// Mitsubishi GX Works2 project: 미니프로젝트6   PLC: Q03UDV

PROGRAM MAIN
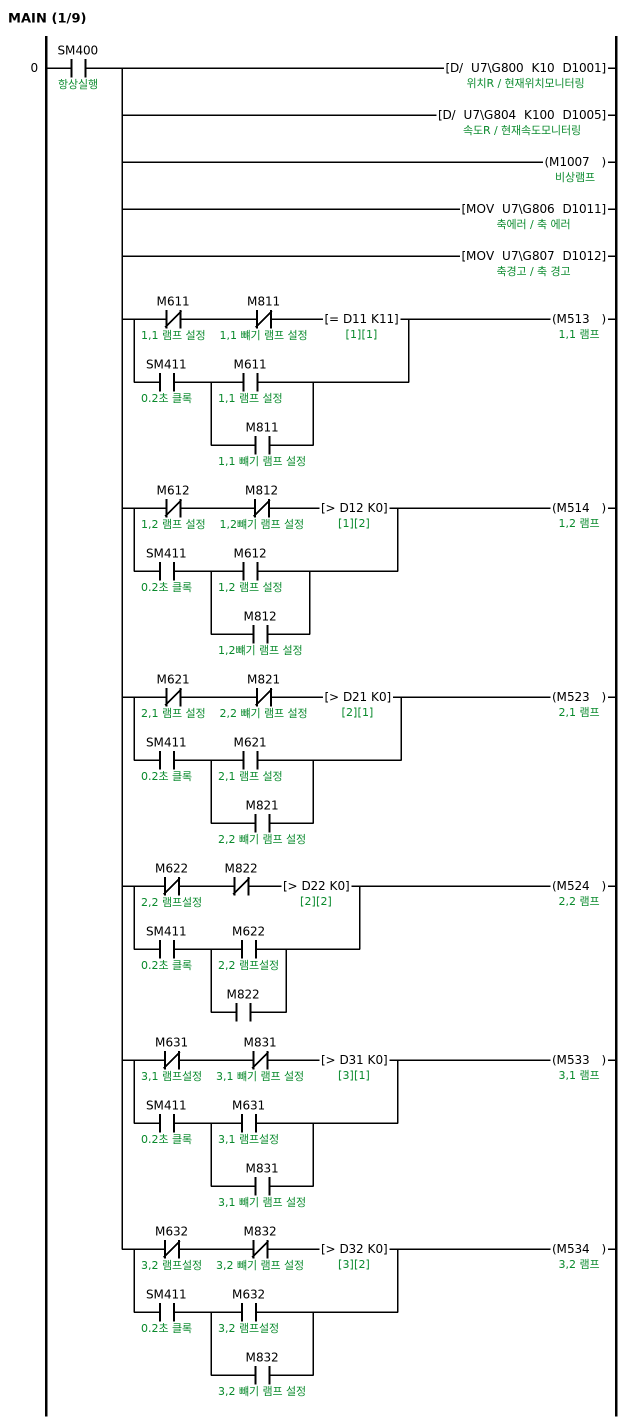
0     LD      SM400  ; 항상실행
      D/      U7\G800 K10 D1001  ; 위치R / 현재위치모니터링
      D/      U7\G804 K100 D1005  ; 속도R / 현재속도모니터링
      OUT     M1007  ; 비상램프
      MOV     U7\G806 D1011  ; 축에러 / 축 에러
      MOV     U7\G807 D1012  ; 축경고 / 축 경고
      MPS
      LDI     M611  ; 1,1 램프 설정
      ANI     M811  ; 1,1 뺴기 램프 설정
      AND=    D11 K11  ; [1][1]
      LD      SM411  ; 0.2초 클록
      LD      M611  ; 1,1 램프 설정
      OR      M811  ; 1,1 뺴기 램프 설정
      ANB
      ORB
      ANB
      OUT     M513  ; 1,1 램프
      MRD
      LDI     M612  ; 1,2 램프 설정
      ANI     M812  ; 1,2뺴기 램프 설정
      AND>    D12 K0  ; [1][2]
      LD      SM411  ; 0.2초 클록
      LD      M612  ; 1,2 램프 설정
      OR      M812  ; 1,2뺴기 램프 설정
      ANB
      ORB
      ANB
      OUT     M514  ; 1,2 램프
      MRD
      LDI     M621  ; 2,1 램프 설정
      ANI     M821  ; 2,2 뺴기 램프 설정
      AND>    D21 K0  ; [2][1]
      LD      SM411  ; 0.2초 클록
      LD      M621  ; 2,1 램프 설정
      OR      M821  ; 2,2 뺴기 램프 설정
      ANB
      ORB
      ANB
      OUT     M523  ; 2,1 램프
      MRD
      LDI     M622  ; 2,2 램프설정
      ANI     M822
      AND>    D22 K0  ; [2][2]
      LD      SM411  ; 0.2초 클록
      LD      M622  ; 2,2 램프설정
      OR      M822
      ANB
      ORB
      ANB
      OUT     M524  ; 2,2 램프
      MRD
      LDI     M631  ; 3,1 램프설정
      ANI     M831  ; 3,1 뺴기 램프 설정
      AND>    D31 K0  ; [3][1]
      LD      SM411  ; 0.2초 클록
      LD      M631  ; 3,1 램프설정
      OR      M831  ; 3,1 뺴기 램프 설정
      ANB
      ORB
      ANB
      OUT     M533  ; 3,1 램프
      MPP
      LDI     M632  ; 3,2 램프설정
      ANI     M832  ; 3,2 뺴기 램프 설정
      AND>    D32 K0  ; [3][2]
      LD      SM411  ; 0.2초 클록
      LD      M632  ; 3,2 램프설정
      OR      M832  ; 3,2 뺴기 램프 설정
      ANB
      ORB
      ANB
      OUT     M534  ; 3,2 램프
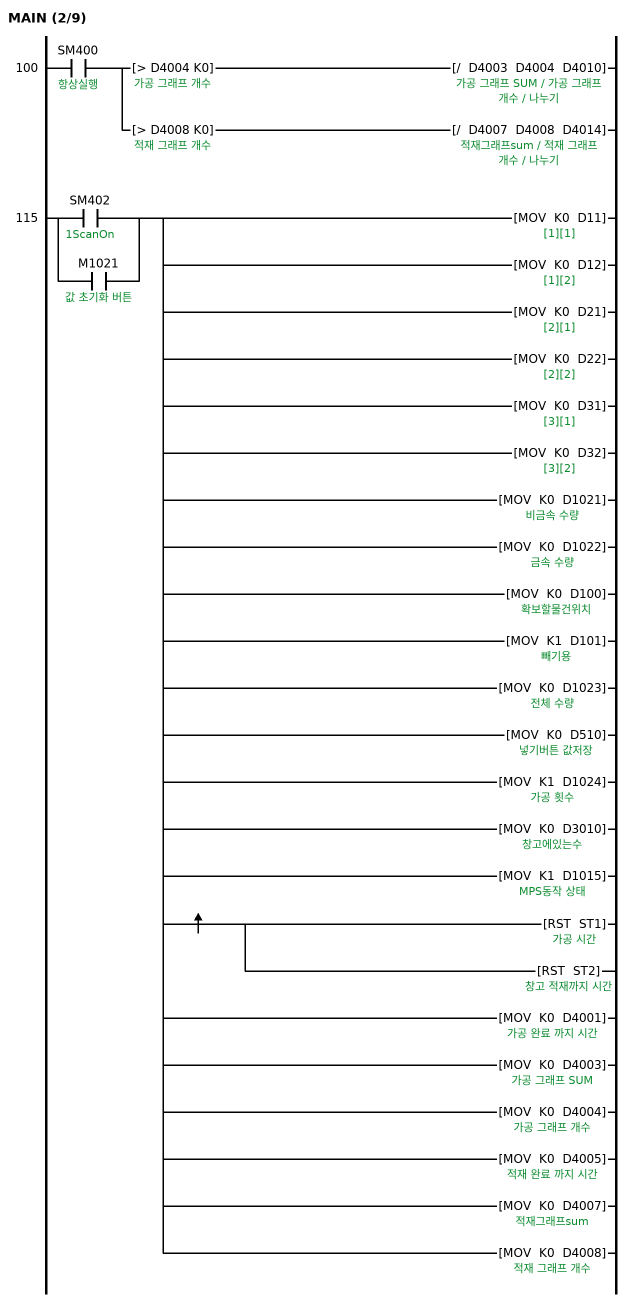
100   LD      SM400  ; 항상실행
      MPS
      AND>    D4004 K0  ; 가공 그래프 개수
      /       D4003 D4004 D4010  ; 가공 그래프 SUM / 나누기
      MPP
      AND>    D4008 K0  ; 적재 그래프 개수
      /       D4007 D4008 D4014  ; 적재그래프sum / 나누기
115   LD      SM402  ; 1ScanOn
      OR      M1021  ; 값 초기화 버튼
      MOV     K0 D11
      MOV     K0 D12
      MOV     K0 D21
      MOV     K0 D22
      MOV     K0 D31
      MOV     K0 D32
      MOV     K0 D1021  ; 비금속 수량
      MOV     K0 D1022  ; 금속 수량
      MOV     K0 D100  ; 확보할물건위치
      MOV     K1 D101  ; 빼기용
      MOV     K0 D1023  ; 전체 수량
      MOV     K0 D510  ; 넣기버튼 값저장
      MOV     K1 D1024  ; 가공 횟수
      MOV     K0 D3010  ; 창고에있는수
      MOV     K1 D1015  ; MPS동작 상태
      MPS
      MEP
      RST     ST1  ; 가공 시간
      RST     ST2  ; 창고 적재까지 시간
      MPP
      MOV     K0 D4001  ; 가공 완료 까지 시간
      MOV     K0 D4003
      MOV     K0 D4004
      MOV     K0 D4005  ; 적재 완료 까지 시간
      MOV     K0 D4007
      MOV     K0 D4008
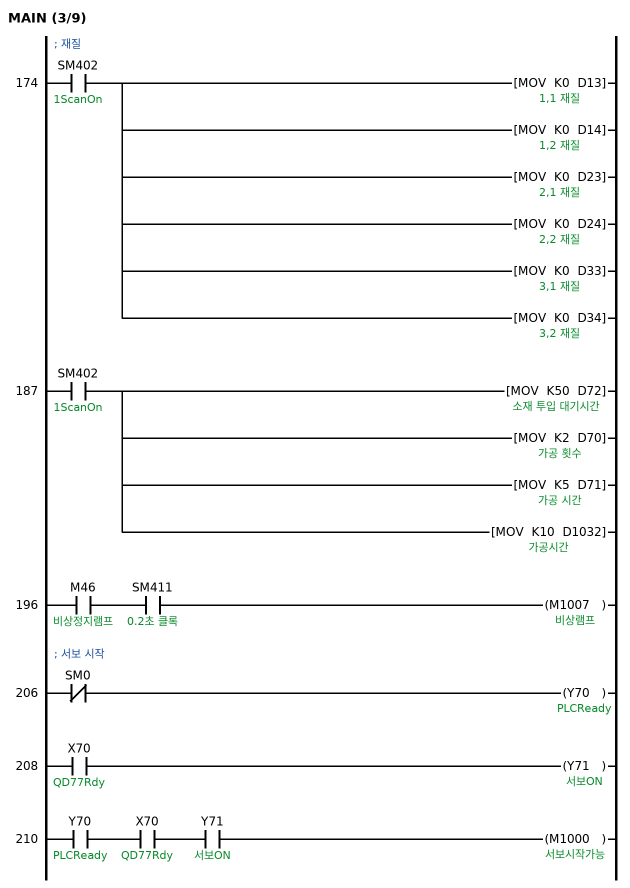
; 재질
174   LD      SM402  ; 1ScanOn
      MOV     K0 D13  ; 1,1 재질
      MOV     K0 D14  ; 1,2 재질
      MOV     K0 D23  ; 2,1 재질
      MOV     K0 D24  ; 2,2 재질
      MOV     K0 D33  ; 3,1 재질
      MOV     K0 D34  ; 3,2 재질
187   LD      SM402  ; 1ScanOn
      MOV     K50 D72  ; 소재 투입 대기시간
      MOV     K2 D70  ; 가공 횟수
      MOV     K5 D71  ; 가공 시간
      MOV     K10 D1032  ; 가공시간
196   LD      M46  ; 비상정지램프
      AND     SM411  ; 0.2초 클록
      OUT     M1007  ; 비상램프
; 서보 시작
206   LDI     SM0
      OUT     Y70  ; PLCReady
208   LD      X70  ; QD77Rdy
      OUT     Y71  ; 서보ON
210   LD      Y70  ; PLCReady
      AND     X70  ; QD77Rdy
      AND     Y71  ; 서보ON
      OUT     M1000  ; 서보시작가능
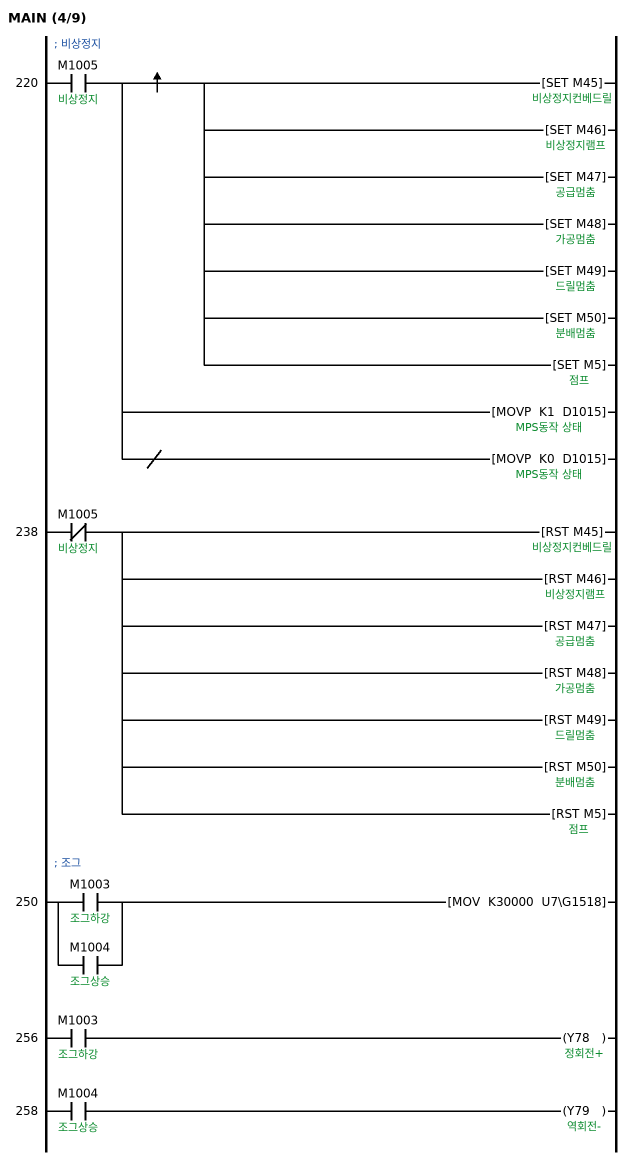
; 비상정지
220   LD      M1005  ; 비상정지
      MPS
      MEP
      SET     M45  ; 비상정지컨베드릴
      SET     M46  ; 비상정지램프
      SET     M47  ; 공급멈춤
      SET     M48  ; 가공멈춤
      SET     M49  ; 드릴멈춤
      SET     M50  ; 분배멈춤
      SET     M5  ; 점프
      MPP
      MOVP    K1 D1015
      INV
      MOVP    K0 D1015
238   LDI     M1005  ; 비상정지
      RST     M45  ; 비상정지컨베드릴
      RST     M46  ; 비상정지램프
      RST     M47  ; 공급멈춤
      RST     M48  ; 가공멈춤
      RST     M49  ; 드릴멈춤
      RST     M50  ; 분배멈춤
      RST     M5  ; 점프
; 조그
250   LD      M1003  ; 조그하강
      OR      M1004  ; 조그상승
      MOV     K30000 U7\G1518
256   LD      M1003  ; 조그하강
      OUT     Y78  ; 정회전+
258   LD      M1004  ; 조그상승
      OUT     Y79  ; 역회전-
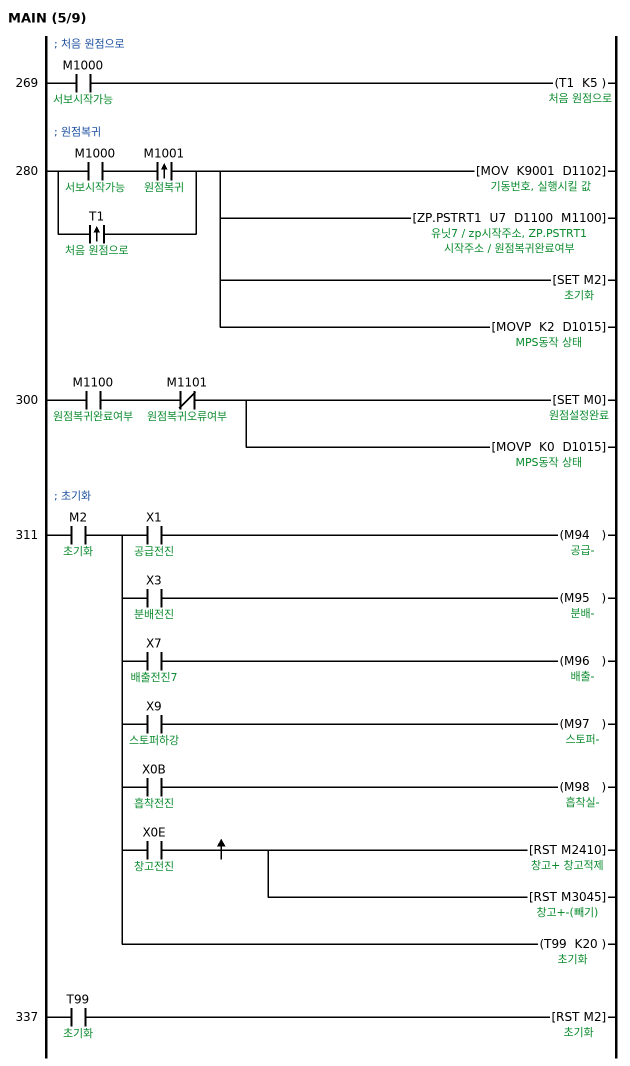
; 처음 원점으로
269   LD      M1000  ; 서보시작가능
      OUT     T1 K5  ; 처음 원점으로
; 원점복귀
280   LD      M1000  ; 서보시작가능
      ANDP    M1001  ; 원점복귀
      ORP     T1  ; 처음 원점으로
      MOV     K9001 D1102  ; 기동번호, 실행시킬 값
      ZP.PSTRT1 U7 D1100 M1100  ; 유닛7 / zp시작주소, ZP.PSTRT1 시작주소 / 원점복귀완료여부
      SET     M2  ; 초기화
      MOVP    K2 D1015
300   LD      M1100  ; 원점복귀완료여부
      ANI     M1101  ; 원점복귀오류여부
      SET     M0  ; 원점설정완료
      MOVP    K0 D1015
; 초기화
311   LD      M2  ; 초기화
      MPS
      AND     X1  ; 공급전진
      OUT     M94  ; 공급-
      MRD
      AND     X3  ; 분배전진
      OUT     M95  ; 분배-
      MRD
      AND     X7  ; 배출전진7
      OUT     M96  ; 배출-
      MRD
      AND     X9  ; 스토퍼하강
      OUT     M97  ; 스토퍼-
      MRD
      AND     X0B  ; 흡착전진
      OUT     M98  ; 흡착실-
      MRD
      AND     X0E  ; 창고전진
      MEP
      RST     M2410  ; 창고+ 창고적제
      RST     M3045  ; 창고+-(빼기)
      MPP
      OUT     T99 K20  ; 초기화
337   LD      T99  ; 초기화
      RST     M2  ; 초기화
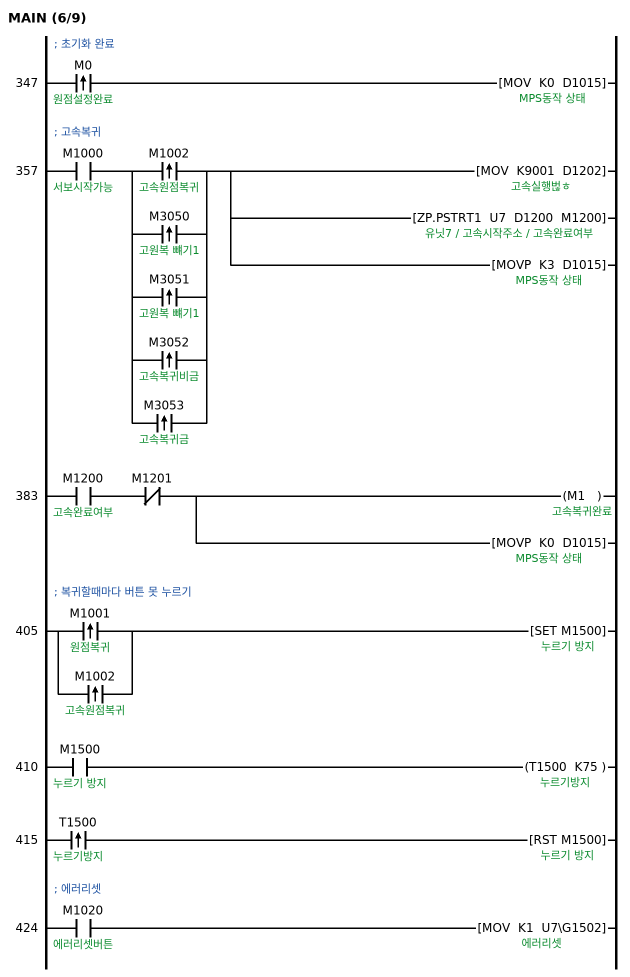
; 초기화 완료
347   LDP     M0  ; 원점설정완료
      MOV     K0 D1015
; 고속복귀
357   LD      M1000  ; 서보시작가능
      LDP     M1002  ; 고속원점복귀
      ORP     M3050  ; 고원복 뺴기1
      ORP     M3051  ; 고원복 뺴기1
      ORP     M3052  ; 고속복귀비금
      ORP     M3053  ; 고속복귀금
      ANB
      MOV     K9001 D1202  ; 고속실행벊ㅎ
      ZP.PSTRT1 U7 D1200 M1200  ; 고속시작주소 / 고속완료여부
      MOVP    K3 D1015
383   LD      M1200  ; 고속완료여부
      ANI     M1201
      OUT     M1  ; 고속복귀완료
      MOVP    K0 D1015
; 복귀할때마다 버튼 못 누르기
405   LDP     M1001  ; 원점복귀
      ORP     M1002  ; 고속원점복귀
      SET     M1500  ; 누르기 방지
410   LD      M1500  ; 누르기 방지
      OUT     T1500 K75  ; 누르기방지
415   LDP     T1500  ; 누르기방지
      RST     M1500  ; 누르기 방지
; 에러리셋
424   LD      M1020  ; 에러리셋버튼
      MOV     K1 U7\G1502  ; 에러리셋
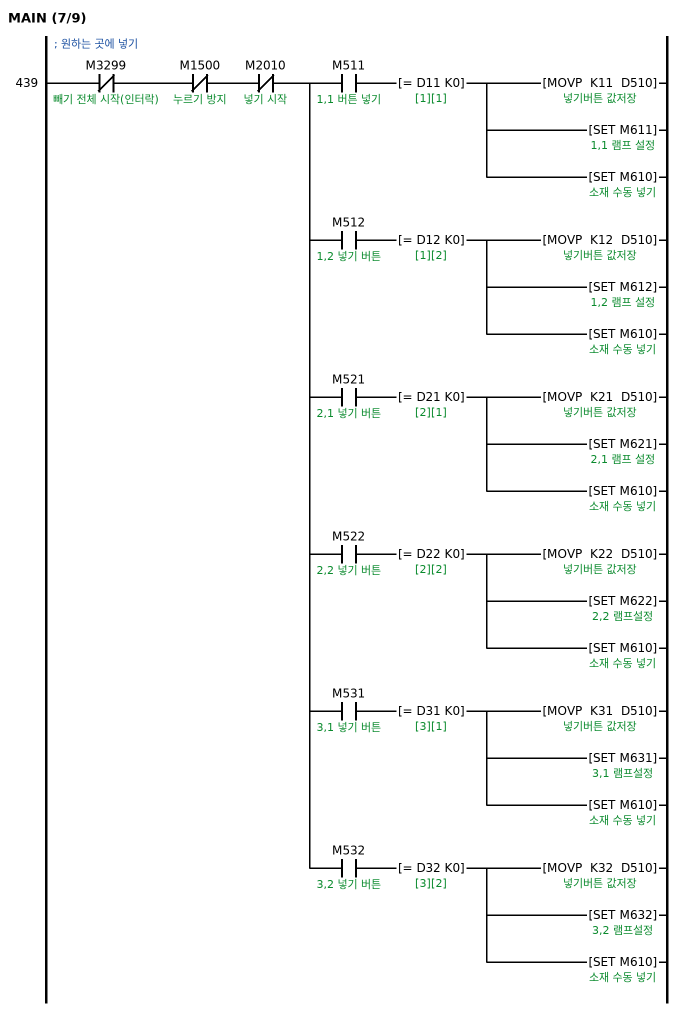
; 원하는 곳에 넣기
439   LDI     M3299  ; 빼기 전체 시작(인터락)
      ANI     M1500  ; 누르기 방지
      ANI     M2010  ; 넣기 시작
      MPS
      AND     M511  ; 1,1 버튼 넣기
      AND=    D11 K0  ; [1][1]
      MOVP    K11 D510
      SET     M611  ; 1,1 램프 설정
      SET     M610  ; 소재 수동 넣기
      MRD
      AND     M512  ; 1,2 넣기 버튼
      AND=    D12 K0  ; [1][2]
      MOVP    K12 D510
      SET     M612  ; 1,2 램프 설정
      SET     M610  ; 소재 수동 넣기
      MRD
      AND     M521  ; 2,1 넣기 버튼
      AND=    D21 K0  ; [2][1]
      MOVP    K21 D510
      SET     M621  ; 2,1 램프 설정
      SET     M610  ; 소재 수동 넣기
      MRD
      AND     M522  ; 2,2 넣기 버튼
      AND=    D22 K0  ; [2][2]
      MOVP    K22 D510
      SET     M622  ; 2,2 램프설정
      SET     M610  ; 소재 수동 넣기
      MRD
      AND     M531  ; 3,1 넣기 버튼
      AND=    D31 K0  ; [3][1]
      MOVP    K31 D510
      SET     M631  ; 3,1 램프설정
      SET     M610  ; 소재 수동 넣기
      MPP
      AND     M532  ; 3,2 넣기 버튼
      AND=    D32 K0  ; [3][2]
      MOVP    K32 D510
      SET     M632  ; 3,2 램프설정
      SET     M610  ; 소재 수동 넣기
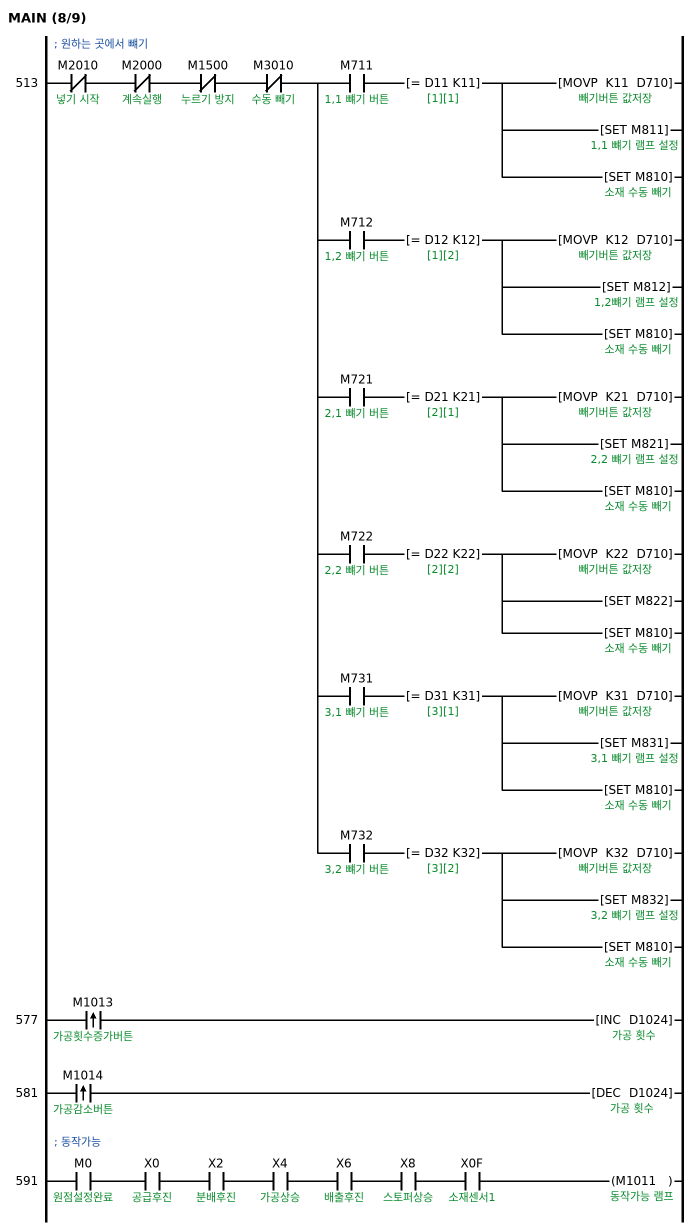
; 원하는 곳에서 뺴기
513   LDI     M2010  ; 넣기 시작
      ANI     M2000  ; 계속실행
      ANI     M1500  ; 누르기 방지
      ANI     M3010  ; 수동 빼기
      MPS
      AND     M711  ; 1,1 뺴기 버튼
      AND=    D11 K11  ; [1][1]
      MOVP    K11 D710  ; 빼기버튼 값저장
      SET     M811  ; 1,1 뺴기 램프 설정
      SET     M810  ; 소재 수동 빼기
      MRD
      AND     M712  ; 1,2 뺴기 버튼
      AND=    D12 K12  ; [1][2]
      MOVP    K12 D710
      SET     M812  ; 1,2뺴기 램프 설정
      SET     M810  ; 소재 수동 빼기
      MRD
      AND     M721  ; 2,1 뺴기 버튼
      AND=    D21 K21  ; [2][1]
      MOVP    K21 D710
      SET     M821  ; 2,2 뺴기 램프 설정
      SET     M810  ; 소재 수동 빼기
      MRD
      AND     M722  ; 2,2 뺴기 버튼
      AND=    D22 K22  ; [2][2]
      MOVP    K22 D710
      SET     M822
      SET     M810  ; 소재 수동 빼기
      MRD
      AND     M731  ; 3,1 뺴기 버튼
      AND=    D31 K31  ; [3][1]
      MOVP    K31 D710
      SET     M831  ; 3,1 뺴기 램프 설정
      SET     M810  ; 소재 수동 빼기
      MPP
      AND     M732  ; 3,2 뺴기 버튼
      AND=    D32 K32  ; [3][2]
      MOVP    K32 D710
      SET     M832  ; 3,2 뺴기 램프 설정
      SET     M810  ; 소재 수동 빼기
577   LDP     M1013  ; 가공횟수증가버튼
      INC     D1024
581   LDP     M1014  ; 가공감소버튼
      DEC     D1024
; 동작가능
591   LD      M0  ; 원점설정완료
      AND     X0  ; 공급후진
      AND     X2  ; 분배후진
      AND     X4  ; 가공상승
      AND     X6  ; 배출후진
      AND     X8  ; 스토퍼상승
      AND     X0F  ; 소재센서1
      OUT     M1011  ; 동작가능 램프
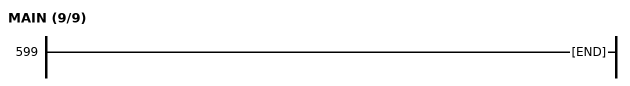
599   END
END_PROGRAM

PROGRAM OUTPUT
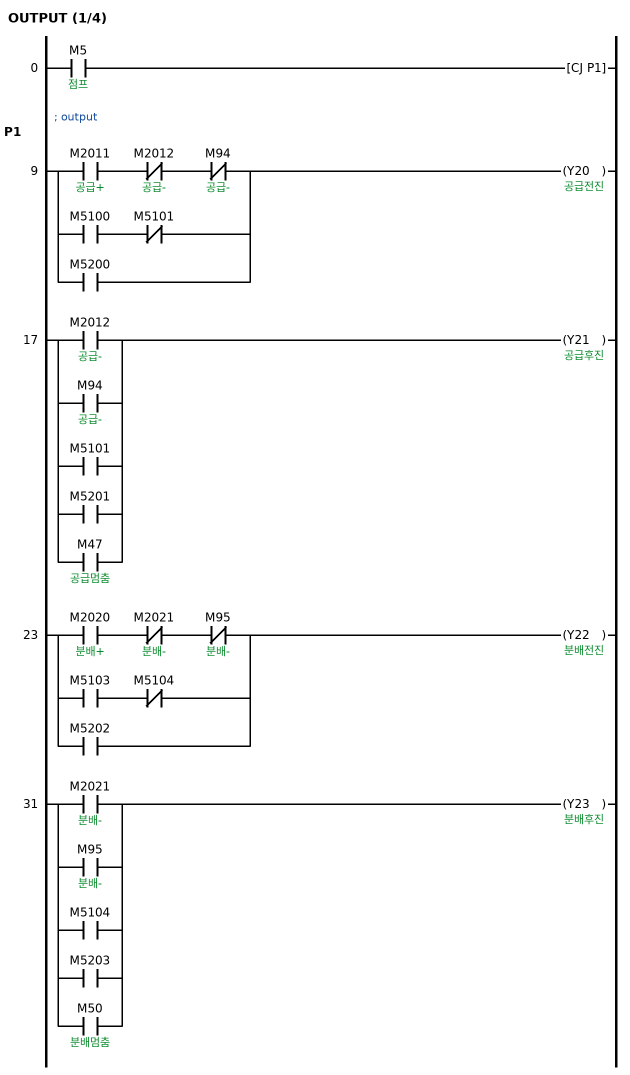
0     LD      M5  ; 점프
      CJ      P1
; output
      P1
9     LD      M2011  ; 공급+
      ANI     M2012  ; 공급-
      ANI     M94  ; 공급-
      LD      M5100
      ANI     M5101
      ORB
      OR      M5200
      OUT     Y20  ; 공급전진
17    LD      M2012  ; 공급-
      OR      M94  ; 공급-
      OR      M5101
      OR      M5201
      OR      M47  ; 공급멈춤
      OUT     Y21  ; 공급후진
23    LD      M2020  ; 분배+
      ANI     M2021  ; 분배-
      ANI     M95  ; 분배-
      LD      M5103
      ANI     M5104
      ORB
      OR      M5202
      OUT     Y22  ; 분배전진
31    LD      M2021  ; 분배-
      OR      M95  ; 분배-
      OR      M5104
      OR      M5203
      OR      M50  ; 분배멈춤
      OUT     Y23  ; 분배후진
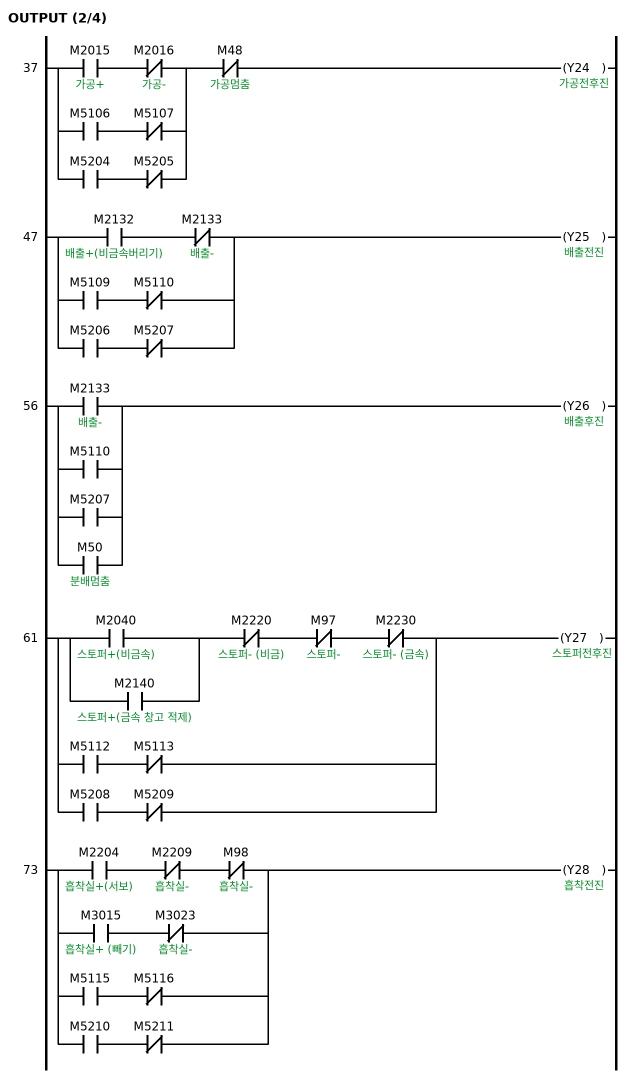
37    LD      M2015  ; 가공+
      ANI     M2016  ; 가공-
      LD      M5106
      ANI     M5107
      ORB
      LD      M5204
      ANI     M5205
      ORB
      ANI     M48  ; 가공멈춤
      OUT     Y24  ; 가공전후진
47    LD      M2132  ; 배출+(비금속버리기)
      ANI     M2133  ; 배출-
      LD      M5109
      ANI     M5110
      ORB
      LD      M5206
      ANI     M5207
      ORB
      OUT     Y25  ; 배출전진
56    LD      M2133  ; 배출-
      OR      M5110
      OR      M5207
      OR      M50  ; 분배멈춤
      OUT     Y26  ; 배출후진
61    LD      M2040  ; 스토퍼+(비금속)
      OR      M2140  ; 스토퍼+(금속 창고 적제)
      ANI     M2220  ; 스토퍼- (비금)
      ANI     M97  ; 스토퍼-
      ANI     M2230  ; 스토퍼- (금속)
      LD      M5112
      ANI     M5113
      ORB
      LD      M5208
      ANI     M5209
      ORB
      OUT     Y27  ; 스토퍼전후진
73    LD      M2204  ; 흡착실+(서보)
      ANI     M2209  ; 흡착실-
      ANI     M98  ; 흡착실-
      LD      M3015  ; 흡착실+ (빼기)
      ANI     M3023  ; 흡착실-
      ORB
      LD      M5115
      ANI     M5116
      ORB
      LD      M5210
      ANI     M5211
      ORB
      OUT     Y28  ; 흡착전진
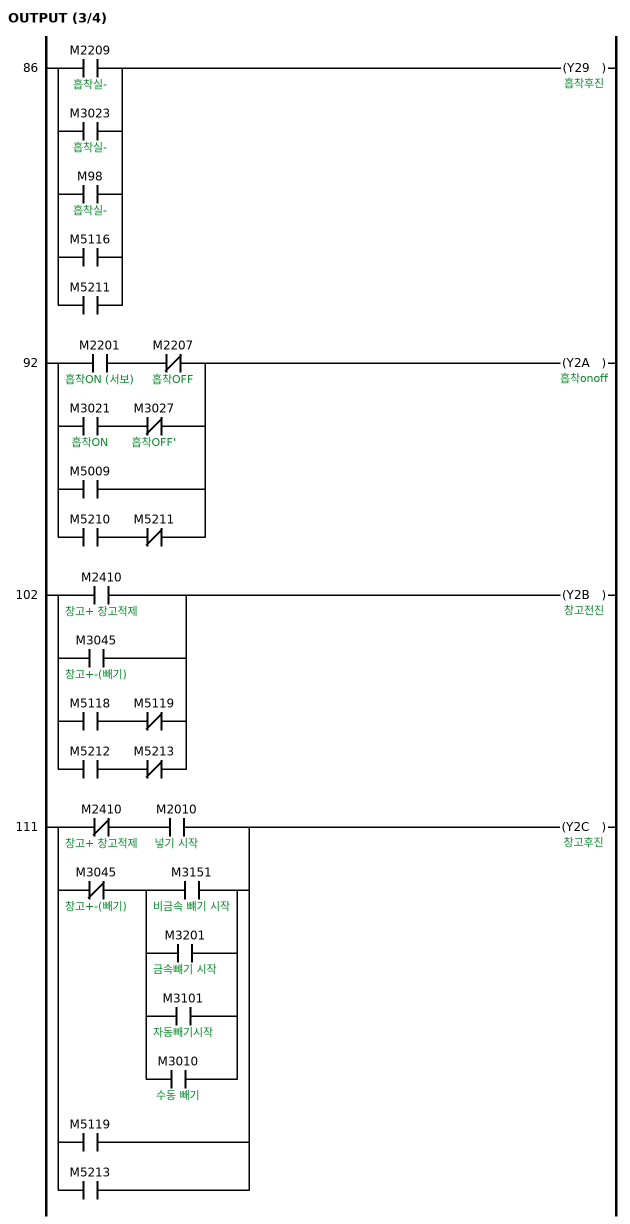
86    LD      M2209  ; 흡착실-
      OR      M3023  ; 흡착실-
      OR      M98  ; 흡착실-
      OR      M5116
      OR      M5211
      OUT     Y29  ; 흡착후진
92    LD      M2201  ; 흡착ON (서보)
      ANI     M2207  ; 흡착OFF
      LD      M3021  ; 흡착ON
      ANI     M3027  ; 흡착OFF'
      ORB
      OR      M5009
      LD      M5210
      ANI     M5211
      ORB
      OUT     Y2A  ; 흡착onoff
102   LD      M2410  ; 창고+ 창고적제
      OR      M3045  ; 창고+-(빼기)
      LD      M5118
      ANI     M5119
      ORB
      LD      M5212
      ANI     M5213
      ORB
      OUT     Y2B  ; 창고전진
111   LDI     M2410  ; 창고+ 창고적제
      AND     M2010  ; 넣기 시작
      LDI     M3045  ; 창고+-(빼기)
      LD      M3151  ; 비금속 뺴기 시작
      OR      M3201  ; 금속뺴기 시작
      OR      M3101  ; 자동빼기시작
      OR      M3010  ; 수동 빼기
      ANB
      ORB
      OR      M5119
      OR      M5213
      OUT     Y2C  ; 창고후진
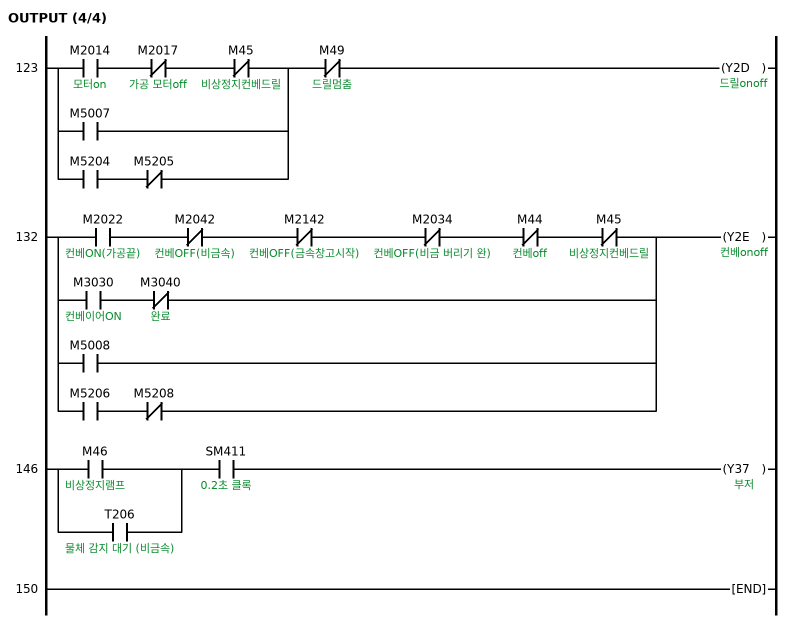
123   LD      M2014  ; 모터on
      ANI     M2017  ; 가공 모터off
      ANI     M45  ; 비상정지컨베드릴
      OR      M5007
      LD      M5204
      ANI     M5205
      ORB
      ANI     M49  ; 드릴멈춤
      OUT     Y2D  ; 드릴onoff
132   LD      M2022  ; 컨베ON(가공끝)
      ANI     M2042  ; 컨베OFF(비금속)
      ANI     M2142  ; 컨베OFF(금속창고시작)
      ANI     M2034  ; 컨베OFF(비금 버리기 완)
      ANI     M44  ; 컨베off
      ANI     M45  ; 비상정지컨베드릴
      LD      M3030  ; 컨베이어ON
      ANI     M3040  ; 완료
      ORB
      OR      M5008
      LD      M5206
      ANI     M5208
      ORB
      OUT     Y2E  ; 컨베onoff
146   LD      M46  ; 비상정지램프
      OR      T206  ; 물체 감지 대기 (비금속)
      AND     SM411  ; 0.2초 클록
      OUT     Y37  ; 부저
150   END
END_PROGRAM

PROGRAM LOADING
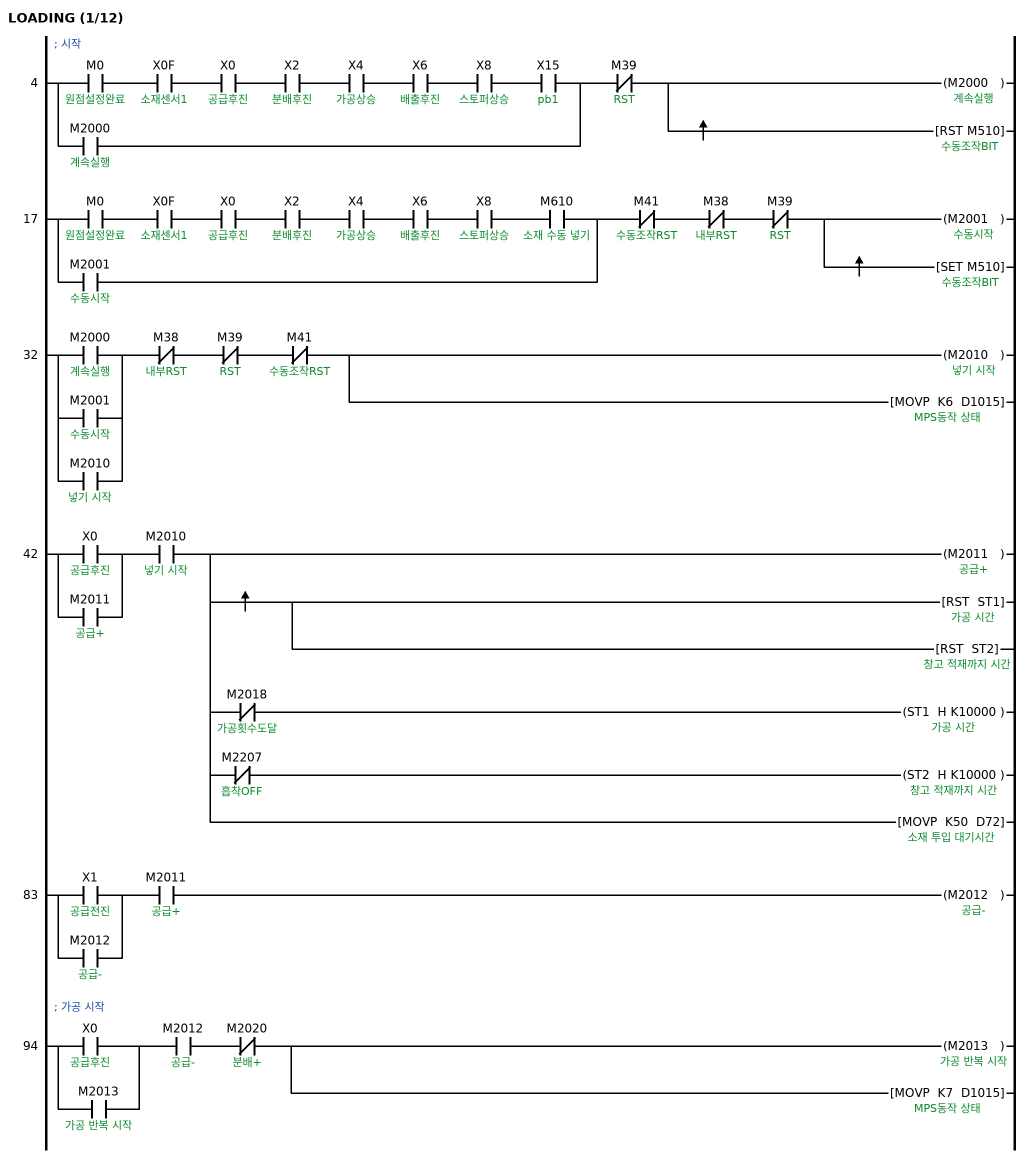
; 시작
4     LD      M0  ; 원점설정완료
      AND     X0F  ; 소재센서1
      AND     X0  ; 공급후진
      AND     X2  ; 분배후진
      AND     X4  ; 가공상승
      AND     X6  ; 배출후진
      AND     X8  ; 스토퍼상승
      AND     X15  ; pb1
      OR      M2000  ; 계속실행
      ANI     M39  ; RST
      OUT     M2000  ; 계속실행
      MEP
      RST     M510  ; 수동조작BIT
17    LD      M0  ; 원점설정완료
      AND     X0F  ; 소재센서1
      AND     X0  ; 공급후진
      AND     X2  ; 분배후진
      AND     X4  ; 가공상승
      AND     X6  ; 배출후진
      AND     X8  ; 스토퍼상승
      AND     M610  ; 소재 수동 넣기
      OR      M2001  ; 수동시작
      ANI     M41  ; 수동조작RST
      ANI     M38  ; 내부RST
      ANI     M39  ; RST
      OUT     M2001  ; 수동시작
      MEP
      SET     M510  ; 수동조작BIT
32    LD      M2000  ; 계속실행
      OR      M2001  ; 수동시작
      OR      M2010  ; 넣기 시작
      ANI     M38  ; 내부RST
      ANI     M39  ; RST
      ANI     M41  ; 수동조작RST
      OUT     M2010  ; 넣기 시작
      MOVP    K6 D1015  ; MPS동작 상태
42    LD      X0  ; 공급후진
      OR      M2011  ; 공급+
      AND     M2010  ; 넣기 시작
      OUT     M2011  ; 공급+
      MPS
      MEP
      RST     ST1  ; 가공 시간
      RST     ST2  ; 창고 적재까지 시간
      MRD
      ANI     M2018  ; 가공횟수도달
      OUTH    ST1 K10000  ; 가공 시간
      MRD
      ANI     M2207  ; 흡착OFF
      OUTH    ST2 K10000  ; 창고 적재까지 시간
      MPP
      MOVP    K50 D72  ; 소재 투입 대기시간
        [note] 5초대기시간 초기화
83    LD      X1  ; 공급전진
      OR      M2012  ; 공급-
      AND     M2011  ; 공급+
      OUT     M2012  ; 공급-
; 가공 시작
94    LD      X0  ; 공급후진
      OR      M2013  ; 가공 반복 시작
      AND     M2012  ; 공급-
      ANI     M2020  ; 분배+
      OUT     M2013  ; 가공 반복 시작
      MOVP    K7 D1015
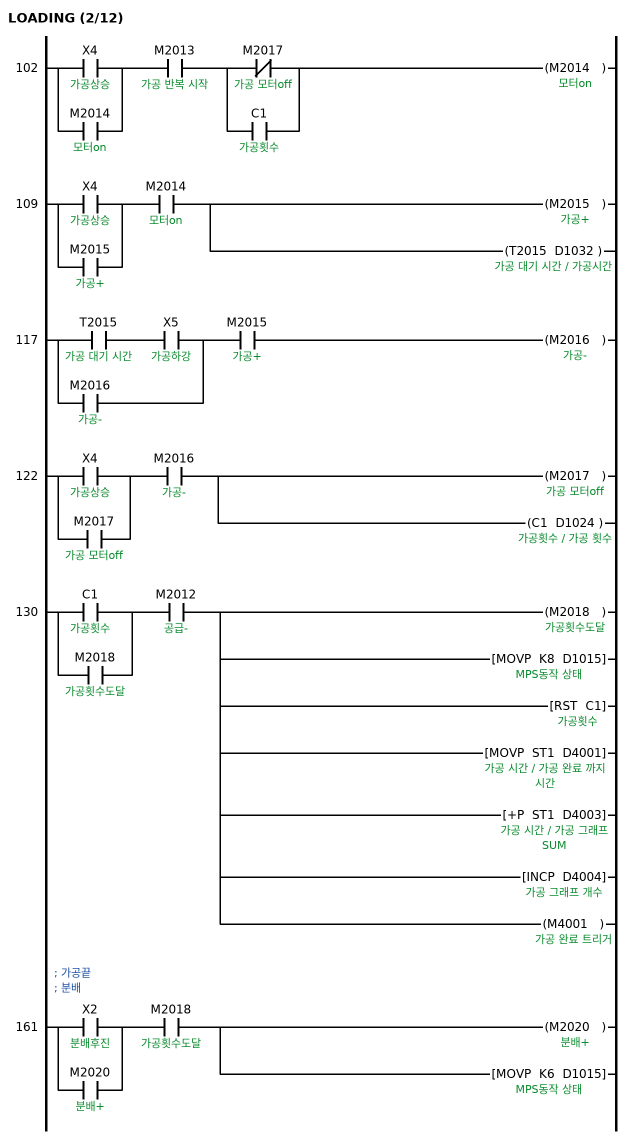
102   LD      X4  ; 가공상승
      OR      M2014  ; 모터on
      AND     M2013  ; 가공 반복 시작
      LDI     M2017  ; 가공 모터off
      OR      C1  ; 가공횟수
      ANB
      OUT     M2014  ; 모터on
109   LD      X4  ; 가공상승
      OR      M2015  ; 가공+
      AND     M2014  ; 모터on
      OUT     M2015  ; 가공+
      OUT     T2015 D1032  ; 가공 대기 시간 / 가공시간
117   LD      T2015  ; 가공 대기 시간
      AND     X5  ; 가공하강
      OR      M2016  ; 가공-
      AND     M2015  ; 가공+
      OUT     M2016  ; 가공-
122   LD      X4  ; 가공상승
      OR      M2017  ; 가공 모터off
      AND     M2016  ; 가공-
      OUT     M2017  ; 가공 모터off
      OUT     C1 D1024  ; 가공횟수 / 가공 횟수
130   LD      C1  ; 가공횟수
      OR      M2018  ; 가공횟수도달
      AND     M2012  ; 공급-
      OUT     M2018  ; 가공횟수도달
      MOVP    K8 D1015
      RST     C1  ; 가공횟수
      MOVP    ST1 D4001  ; 가공 완료 까지 시간
      +P      ST1 D4003  ; 가공 그래프 SUM
      INCP    D4004  ; 가공 그래프 개수
      OUT     M4001  ; 가공 완료 트리거
; 가공끝
; 분배
161   LD      X2  ; 분배후진
      OR      M2020  ; 분배+
      AND     M2018  ; 가공횟수도달
      OUT     M2020  ; 분배+
      MOVP    K6 D1015
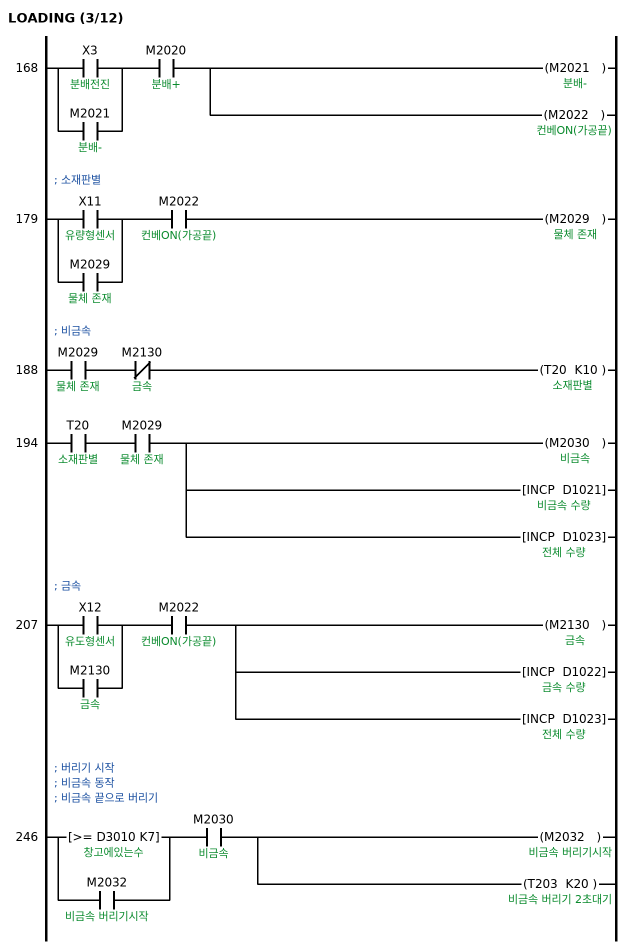
168   LD      X3  ; 분배전진
      OR      M2021  ; 분배-
      AND     M2020  ; 분배+
      OUT     M2021  ; 분배-
      OUT     M2022  ; 컨베ON(가공끝)
; 소재판별
179   LD      X11  ; 유량형센서
      OR      M2029  ; 물체 존재
      AND     M2022  ; 컨베ON(가공끝)
      OUT     M2029  ; 물체 존재
; 비금속
188   LD      M2029  ; 물체 존재
      ANI     M2130  ; 금속
      OUT     T20 K10  ; 소재판별
194   LD      T20  ; 소재판별
      AND     M2029  ; 물체 존재
      OUT     M2030  ; 비금속
      INCP    D1021  ; 비금속 수량
      INCP    D1023  ; 전체 수량
; 금속
207   LD      X12  ; 유도형센서
      OR      M2130  ; 금속
      AND     M2022  ; 컨베ON(가공끝)
      OUT     M2130  ; 금속
      INCP    D1022  ; 금속 수량
      INCP    D1023
; 버리기 시작
; 비금속 동작
; 비금속 끝으로 버리기
246   LD>=    D3010 K7  ; 창고에있는수
      OR      M2032  ; 비금속 버리기시작
      AND     M2030  ; 비금속
      OUT     M2032  ; 비금속 버리기시작
      OUT     T203 K20  ; 비금속 버리기 2초대기
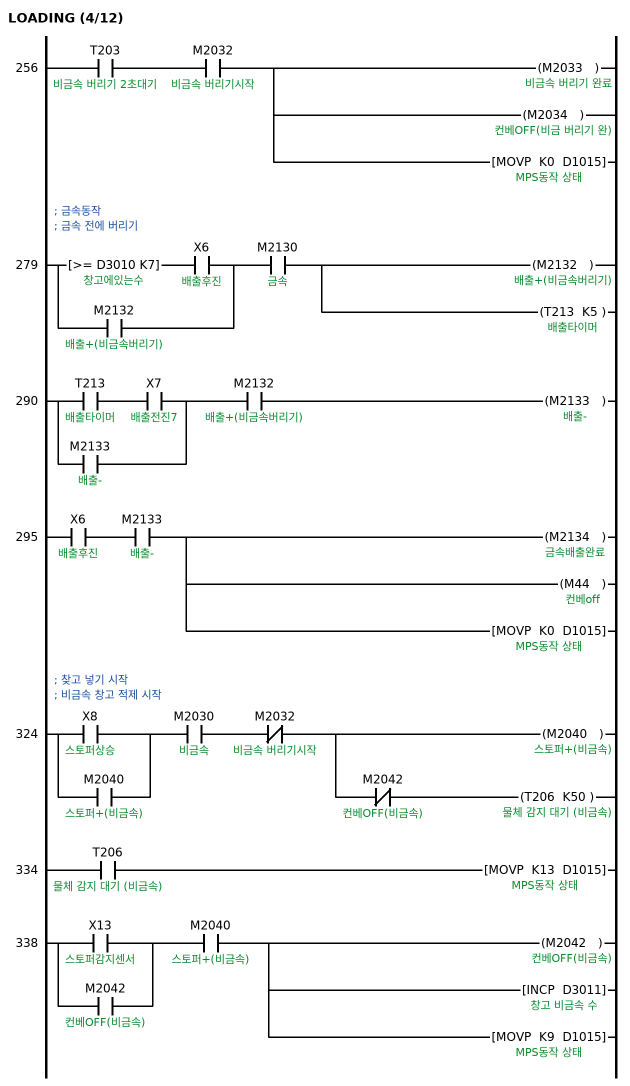
256   LD      T203  ; 비금속 버리기 2초대기
      AND     M2032  ; 비금속 버리기시작
      OUT     M2033  ; 비금속 버리기 완료
      OUT     M2034  ; 컨베OFF(비금 버리기 완)
      MOVP    K0 D1015
; 금속동작
; 금속 전에 버리기
279   LD>=    D3010 K7  ; 창고에있는수
      AND     X6  ; 배출후진
      OR      M2132  ; 배출+(비금속버리기)
      AND     M2130  ; 금속
      OUT     M2132  ; 배출+(비금속버리기)
      OUT     T213 K5  ; 배출타이머
290   LD      T213  ; 배출타이머
      AND     X7  ; 배출전진7
      OR      M2133  ; 배출-
      AND     M2132  ; 배출+(비금속버리기)
      OUT     M2133  ; 배출-
295   LD      X6  ; 배출후진
      AND     M2133  ; 배출-
      OUT     M2134  ; 금속배출완료
      OUT     M44  ; 컨베off
      MOVP    K0 D1015
; 찾고 넣기 시작
; 비금속 창고 적제 시작
324   LD      X8  ; 스토퍼상승
      OR      M2040  ; 스토퍼+(비금속)
      AND     M2030  ; 비금속
      ANI     M2032  ; 비금속 버리기시작
      OUT     M2040  ; 스토퍼+(비금속)
      ANI     M2042  ; 컨베OFF(비금속)
      OUT     T206 K50  ; 물체 감지 대기 (비금속)
334   LD      T206  ; 물체 감지 대기 (비금속)
      MOVP    K13 D1015
338   LD      X13  ; 스토퍼감지센서
      OR      M2042  ; 컨베OFF(비금속)
      AND     M2040  ; 스토퍼+(비금속)
      OUT     M2042  ; 컨베OFF(비금속)
      INCP    D3011  ; 창고 비금속 수
      MOVP    K9 D1015
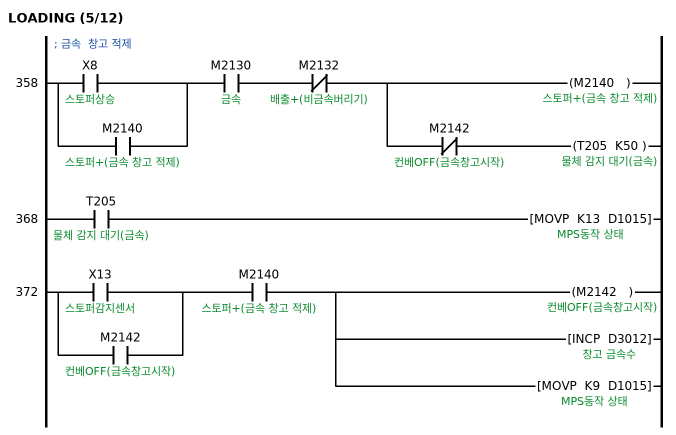
; 금속  창고 적제
358   LD      X8  ; 스토퍼상승
      OR      M2140  ; 스토퍼+(금속 창고 적제)
      AND     M2130  ; 금속
      ANI     M2132  ; 배출+(비금속버리기)
      OUT     M2140  ; 스토퍼+(금속 창고 적제)
      ANI     M2142  ; 컨베OFF(금속창고시작)
      OUT     T205 K50  ; 물체 감지 대기(금속)
368   LD      T205  ; 물체 감지 대기(금속)
      MOVP    K13 D1015
372   LD      X13  ; 스토퍼감지센서
      OR      M2142  ; 컨베OFF(금속창고시작)
      AND     M2140  ; 스토퍼+(금속 창고 적제)
      OUT     M2142  ; 컨베OFF(금속창고시작)
      INCP    D3012  ; 창고 금속수
      MOVP    K9 D1015
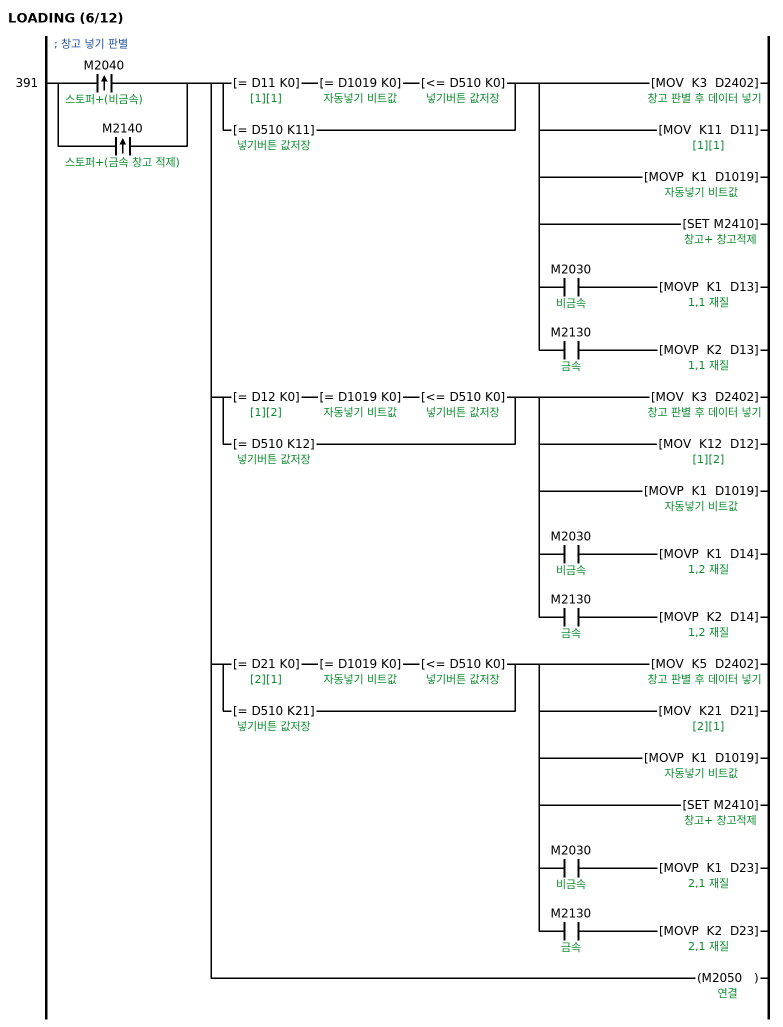
; 창고 넣기 판별
391   LDP     M2040  ; 스토퍼+(비금속)
      ORP     M2140  ; 스토퍼+(금속 창고 적제)
      MPS
      LD=     D11 K0  ; [1][1]
      AND=    D1019 K0  ; 자동넣기 비트값
      AND<=   D510 K0  ; 넣기버튼 값저장
      OR=     D510 K11  ; 넣기버튼 값저장
      ANB
      MOV     K3 D2402  ; 창고 판별 후 데이터 넣기
      MOV     K11 D11
      MOVP    K1 D1019
      SET     M2410  ; 창고+ 창고적제
      MPS
      AND     M2030  ; 비금속
      MOVP    K1 D13  ; 1,1 재질
      MPP
      AND     M2130  ; 금속
      MOVP    K2 D13
      MRD
      LD=     D12 K0  ; [1][2]
      AND=    D1019 K0  ; 자동넣기 비트값
      AND<=   D510 K0  ; 넣기버튼 값저장
      OR=     D510 K12  ; 넣기버튼 값저장
      ANB
      MOV     K3 D2402
      MOV     K12 D12
      MOVP    K1 D1019
      MPS
      AND     M2030  ; 비금속
      MOVP    K1 D14  ; 1,2 재질
      MPP
      AND     M2130  ; 금속
      MOVP    K2 D14
      MRD
      LD=     D21 K0  ; [2][1]
      AND=    D1019 K0  ; 자동넣기 비트값
      AND<=   D510 K0  ; 넣기버튼 값저장
      OR=     D510 K21  ; 넣기버튼 값저장
      ANB
      MOV     K5 D2402
      MOV     K21 D21
      MOVP    K1 D1019
      SET     M2410  ; 창고+ 창고적제
      MPS
      AND     M2030  ; 비금속
      MOVP    K1 D23  ; 2,1 재질
      MPP
      AND     M2130  ; 금속
      MOVP    K2 D23
      MPP
      OUT     M2050  ; 연결
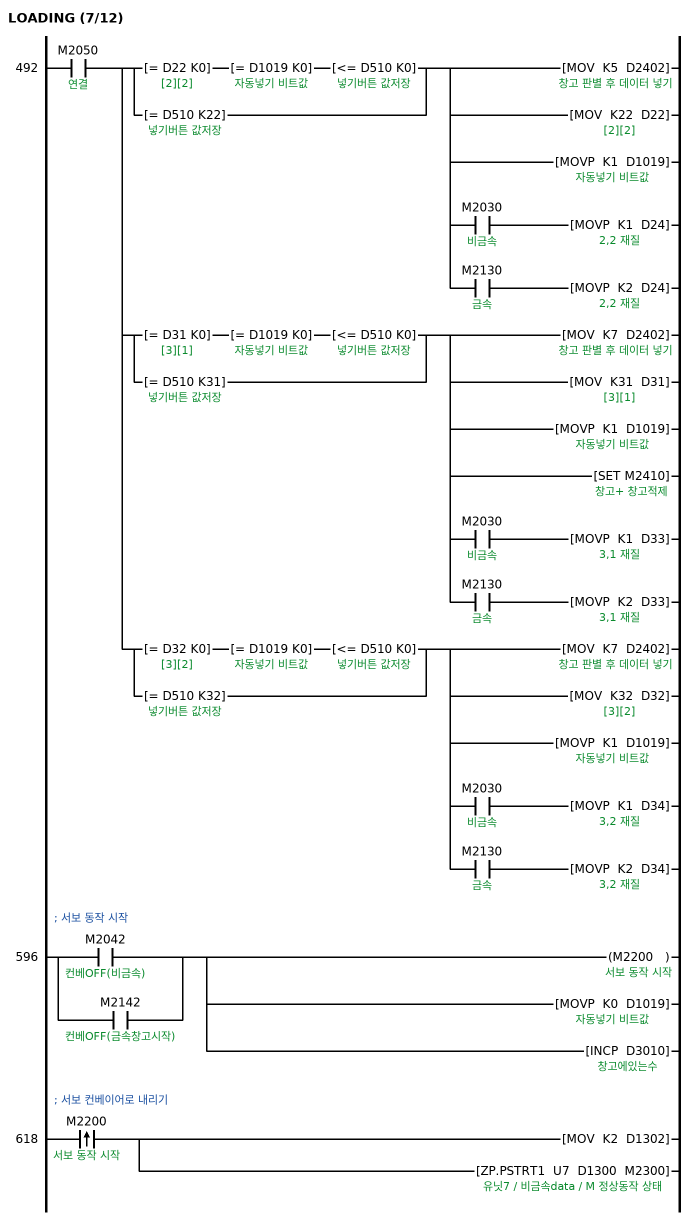
492   LD      M2050  ; 연결
      MPS
      LD=     D22 K0  ; [2][2]
      AND=    D1019 K0  ; 자동넣기 비트값
      AND<=   D510 K0  ; 넣기버튼 값저장
      OR=     D510 K22  ; 넣기버튼 값저장
      ANB
      MOV     K5 D2402
      MOV     K22 D22
      MOVP    K1 D1019
      MPS
      AND     M2030  ; 비금속
      MOVP    K1 D24  ; 2,2 재질
      MPP
      AND     M2130  ; 금속
      MOVP    K2 D24
      MRD
      LD=     D31 K0  ; [3][1]
      AND=    D1019 K0  ; 자동넣기 비트값
      AND<=   D510 K0  ; 넣기버튼 값저장
      OR=     D510 K31  ; 넣기버튼 값저장
      ANB
      MOV     K7 D2402
      MOV     K31 D31
      MOVP    K1 D1019
      SET     M2410  ; 창고+ 창고적제
      MPS
      AND     M2030  ; 비금속
      MOVP    K1 D33  ; 3,1 재질
      MPP
      AND     M2130  ; 금속
      MOVP    K2 D33
      MPP
      LD=     D32 K0  ; [3][2]
      AND=    D1019 K0  ; 자동넣기 비트값
      AND<=   D510 K0  ; 넣기버튼 값저장
      OR=     D510 K32  ; 넣기버튼 값저장
      ANB
      MOV     K7 D2402
      MOV     K32 D32
      MOVP    K1 D1019
      MPS
      AND     M2030  ; 비금속
      MOVP    K1 D34  ; 3,2 재질
      MPP
      AND     M2130  ; 금속
      MOVP    K2 D34
; 서보 동작 시작
596   LD      M2042  ; 컨베OFF(비금속)
      OR      M2142  ; 컨베OFF(금속창고시작)
      OUT     M2200  ; 서보 동작 시작
      MOVP    K0 D1019
      INCP    D3010
; 서보 컨베이어로 내리기
618   LDP     M2200  ; 서보 동작 시작
      MOV     K2 D1302
      ZP.PSTRT1 U7 D1300 M2300  ; 유닛7 / 비금속data / M 정상동작 상태
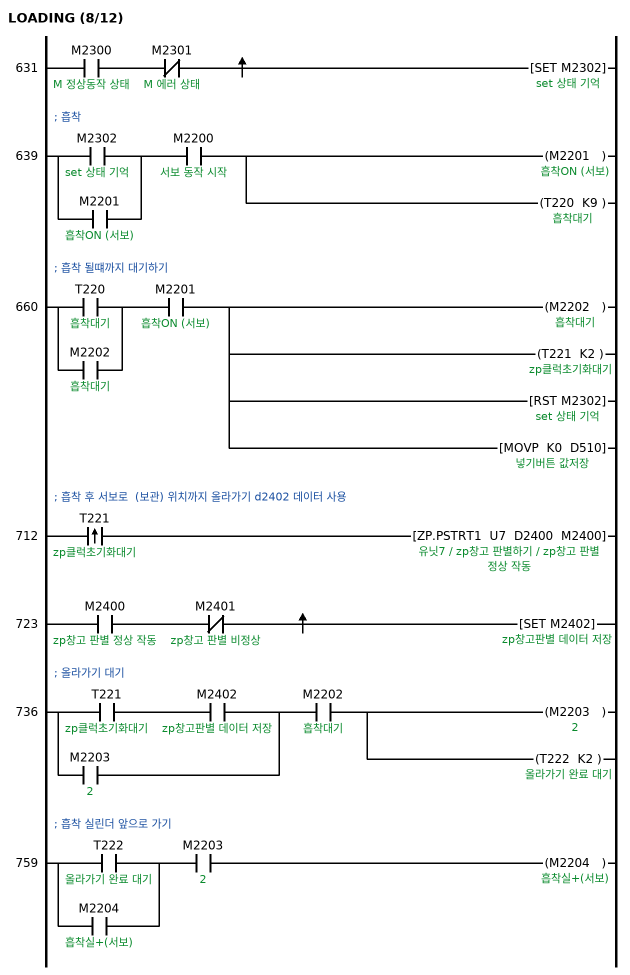
631   LD      M2300  ; M 정상동작 상태
      ANI     M2301  ; M 에러 상태
      MEP
      SET     M2302  ; set 상태 기억
; 흡착
639   LD      M2302  ; set 상태 기억
      OR      M2201  ; 흡착ON (서보)
      AND     M2200  ; 서보 동작 시작
      OUT     M2201  ; 흡착ON (서보)
      OUT     T220 K9  ; 흡착대기
; 흡착 될떄까지 대기하기
660   LD      T220  ; 흡착대기
      OR      M2202  ; 흡착대기
      AND     M2201  ; 흡착ON (서보)
      OUT     M2202  ; 흡착대기
      OUT     T221 K2  ; zp클럭초기화대기
      RST     M2302  ; set 상태 기억
      MOVP    K0 D510
        [note] 넣기값 초기화
; 흡착 후 서보로  (보관) 위치까지 올라가기 d2402 데이터 사용
712   LDP     T221  ; zp클럭초기화대기
      ZP.PSTRT1 U7 D2400 M2400  ; zp창고 판별하기 / zp창고 판별 정상 작동
723   LD      M2400  ; zp창고 판별 정상 작동
      ANI     M2401  ; zp창고 판별 비정상
      MEP
      SET     M2402  ; zp창고판별 데이터 저장
; 올라가기 대기
736   LD      T221  ; zp클럭초기화대기
      AND     M2402  ; zp창고판별 데이터 저장
      OR      M2203  ; 2
      AND     M2202  ; 흡착대기
      OUT     M2203  ; 2
      OUT     T222 K2  ; 올라가기 완료 대기
; 흡착 실린더 앞으로 가기
759   LD      T222  ; 올라가기 완료 대기
      OR      M2204  ; 흡착실+(서보)
      AND     M2203  ; 2
      OUT     M2204  ; 흡착실+(서보)
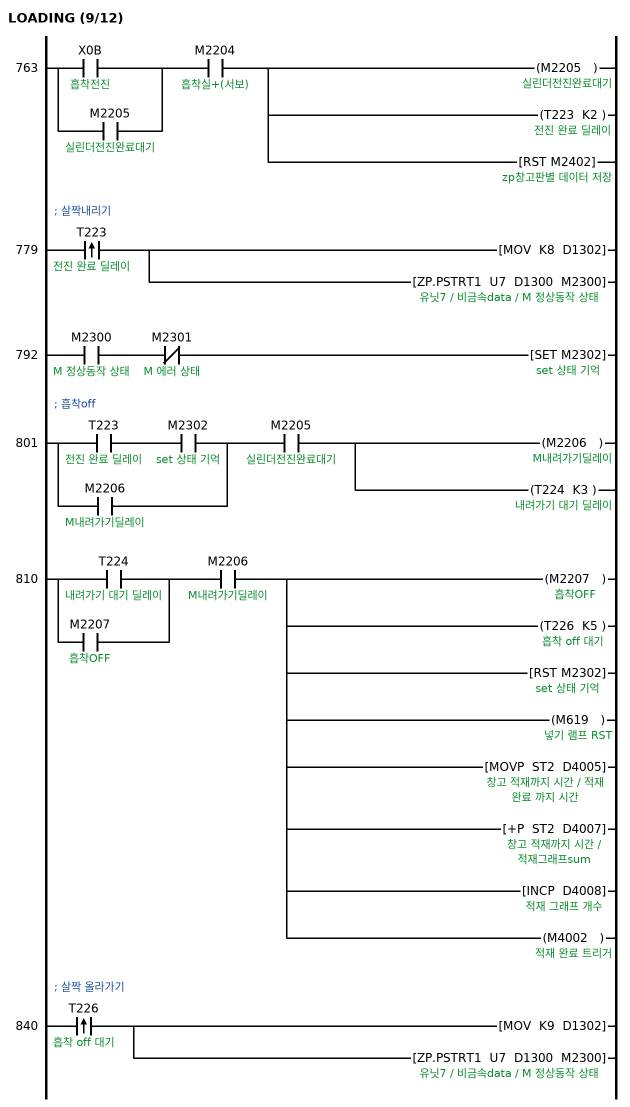
763   LD      X0B  ; 흡착전진
      OR      M2205  ; 실린더전진완료대기
      AND     M2204  ; 흡착실+(서보)
      OUT     M2205  ; 실린더전진완료대기
      OUT     T223 K2  ; 전진 완료 딜레이
      RST     M2402  ; zp창고판별 데이터 저장
; 살짝내리기
779   LDP     T223  ; 전진 완료 딜레이
      MOV     K8 D1302
      ZP.PSTRT1 U7 D1300 M2300
792   LD      M2300  ; M 정상동작 상태
      ANI     M2301  ; M 에러 상태
      SET     M2302  ; set 상태 기억
; 흡착off
801   LD      T223  ; 전진 완료 딜레이
      AND     M2302  ; set 상태 기억
      OR      M2206  ; M내려가기딜레이
      AND     M2205  ; 실린더전진완료대기
      OUT     M2206  ; M내려가기딜레이
      OUT     T224 K3  ; 내려가기 대기 딜레이
810   LD      T224  ; 내려가기 대기 딜레이
      OR      M2207  ; 흡착OFF
      AND     M2206  ; M내려가기딜레이
      OUT     M2207  ; 흡착OFF
      OUT     T226 K5  ; 흡착 off 대기
      RST     M2302  ; set 상태 기억
      OUT     M619  ; 넣기 램프 RST
      MOVP    ST2 D4005  ; 적재 완료 까지 시간
      +P      ST2 D4007  ; 적재그래프sum
      INCP    D4008  ; 적재 그래프 개수
      OUT     M4002  ; 적재 완료 트리거
; 살짝 올라가기
840   LDP     T226  ; 흡착 off 대기
      MOV     K9 D1302
      ZP.PSTRT1 U7 D1300 M2300
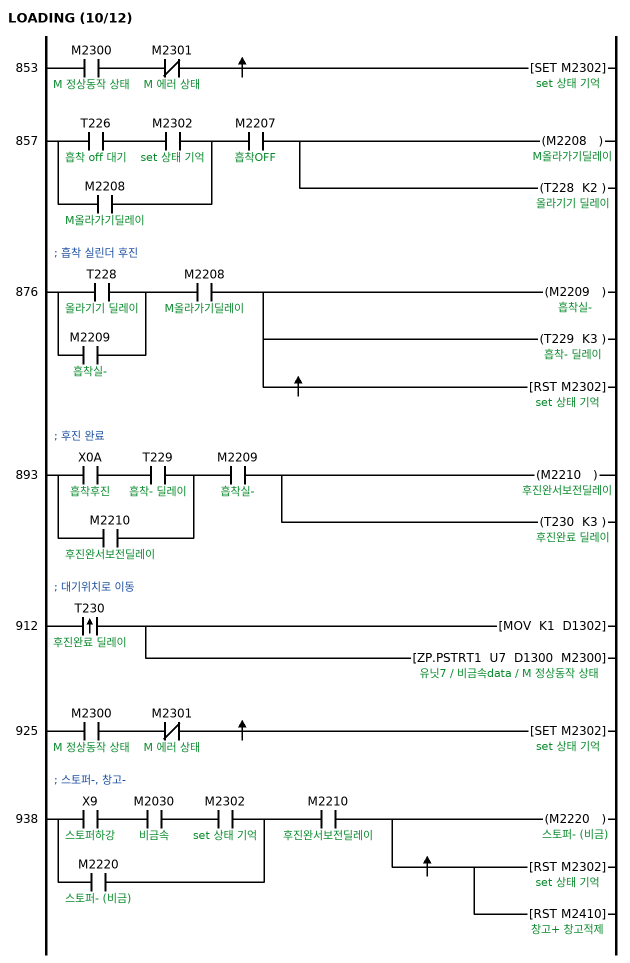
853   LD      M2300  ; M 정상동작 상태
      ANI     M2301  ; M 에러 상태
      MEP
      SET     M2302  ; set 상태 기억
857   LD      T226  ; 흡착 off 대기
      AND     M2302  ; set 상태 기억
      OR      M2208  ; M올라가기딜레이
      AND     M2207  ; 흡착OFF
      OUT     M2208  ; M올라가기딜레이
      OUT     T228 K2  ; 올라기기 딜레이
; 흡착 실린더 후진
876   LD      T228  ; 올라기기 딜레이
      OR      M2209  ; 흡착실-
      AND     M2208  ; M올라가기딜레이
      OUT     M2209  ; 흡착실-
      OUT     T229 K3  ; 흡착- 딜레이
      MEP
      RST     M2302  ; set 상태 기억
; 후진 완료
893   LD      X0A  ; 흡착후진
      AND     T229  ; 흡착- 딜레이
      OR      M2210  ; 후진완서보전딜레이
      AND     M2209  ; 흡착실-
      OUT     M2210  ; 후진완서보전딜레이
      OUT     T230 K3  ; 후진완료 딜레이
; 대기위치로 이동
912   LDP     T230  ; 후진완료 딜레이
      MOV     K1 D1302
      ZP.PSTRT1 U7 D1300 M2300
925   LD      M2300  ; M 정상동작 상태
      ANI     M2301  ; M 에러 상태
      MEP
      SET     M2302  ; set 상태 기억
; 스토퍼-, 창고-
938   LD      X9  ; 스토퍼하강
      AND     M2030  ; 비금속
      AND     M2302  ; set 상태 기억
      OR      M2220  ; 스토퍼- (비금)
      AND     M2210  ; 후진완서보전딜레이
      OUT     M2220  ; 스토퍼- (비금)
      MEP
      RST     M2302  ; set 상태 기억
      RST     M2410  ; 창고+ 창고적제
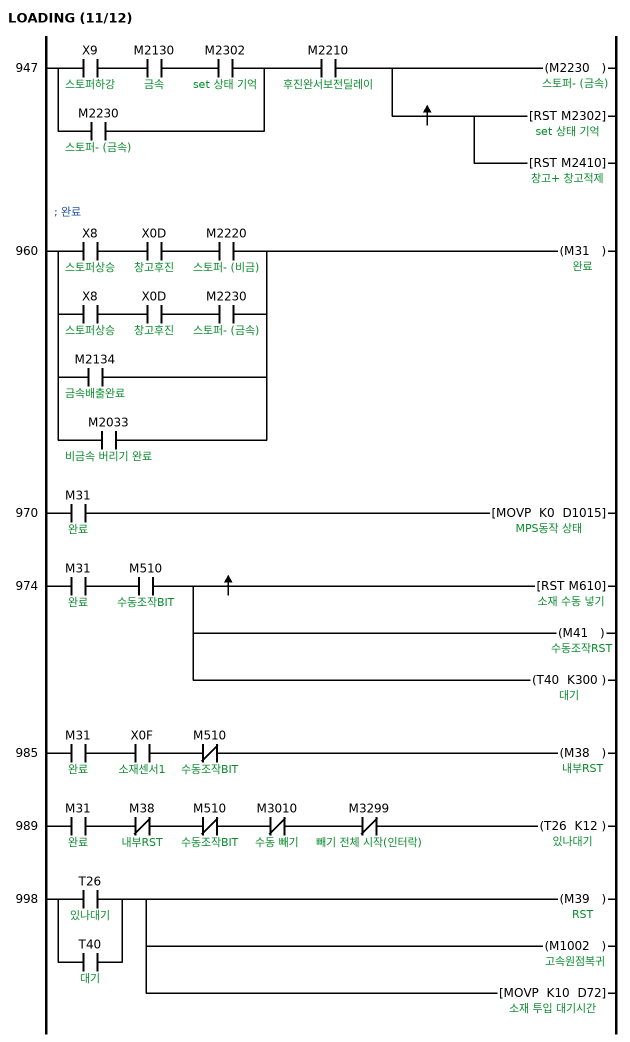
947   LD      X9  ; 스토퍼하강
      AND     M2130  ; 금속
      AND     M2302  ; set 상태 기억
      OR      M2230  ; 스토퍼- (금속)
      AND     M2210  ; 후진완서보전딜레이
      OUT     M2230  ; 스토퍼- (금속)
      MEP
      RST     M2302  ; set 상태 기억
      RST     M2410  ; 창고+ 창고적제
; 완료
960   LD      X8  ; 스토퍼상승
      AND     X0D  ; 창고후진
      AND     M2220  ; 스토퍼- (비금)
      LD      X8  ; 스토퍼상승
      AND     X0D  ; 창고후진
      AND     M2230  ; 스토퍼- (금속)
      ORB
      OR      M2134  ; 금속배출완료
      OR      M2033  ; 비금속 버리기 완료
      OUT     M31  ; 완료
970   LD      M31  ; 완료
      MOVP    K0 D1015
974   LD      M31  ; 완료
      AND     M510  ; 수동조작BIT
      MPS
      MEP
      RST     M610  ; 소재 수동 넣기
      MPP
      OUT     M41  ; 수동조작RST
      OUT     T40 K300  ; 대기
985   LD      M31  ; 완료
      AND     X0F  ; 소재센서1
      ANI     M510  ; 수동조작BIT
      OUT     M38  ; 내부RST
989   LD      M31  ; 완료
      ANI     M38  ; 내부RST
      ANI     M510  ; 수동조작BIT
      ANI     M3010  ; 수동 빼기
      ANI     M3299  ; 빼기 전체 시작(인터락)
      OUT     T26 K12  ; 있나대기
998   LD      T26  ; 있나대기
      OR      T40  ; 대기
      OUT     M39  ; RST
      OUT     M1002  ; 고속원점복귀
      MOVP    K10 D72
